# EPICS autosave request: softGlueApp/Db/QuadDec_settings.req
$(P)$(H)QuadDec-$(N)_A_Signal
$(P)$(H)QuadDec-$(N)_B_Signal
$(P)$(H)QuadDec-$(N)_CLOCK_Signal
$(P)$(H)QuadDec-$(N)_STEP_Signal
$(P)$(H)QuadDec-$(N)_DIR_Signal
$(P)$(H)QuadDec-$(N)_MISS_Signal
$(P)$(H)QuadDec-$(N)_MISSCLR_Signal
